(* CoDeSys 2.3.9.55 project: Test_testLib.pro *)
(* Author: Philip Henriksen *)
(* Libraries: TestLib.lib 13.6.19 08:25:14, Standard.lib 20.5.14 08:13:26, Iecsfc.lib 30.1.13 13:05:12 *)

(* PLC configuration (modules and I/O channels)
K-Bus [K_Bus] node 0, in %IB0 out %QB0 {KbusBusMode = 1; KbusCycleTime = 10000; KbusThreadPriority = 0; KbusSetOutputsToZeroOnApplicationStop = 1}
Modbus variables [PFC200MODBUS] node 1, in %IB0 out %QB0 {PlcStopBehaviour = 1; FiledbusErrorBehaviour = 1; TcpOperation = 1; TcpPort = 502; TcpTimeout = 600; UdpOperation = 1; UdpPort = 502; RtuOperation = 0; NodeId = 1; ResponseTimeout = 100; Interface = 0; Baud = 115200; StopBits = 1; Parity = 1; FlowCtrl = 0; PhysInterface = 0}
Modbus-Master [MB_MASTER] node 2, in %IB0 out %QB0
*)

(* Global variable list: Var_Constant *)
VAR_GLOBAL CONSTANT
	BTFDevice:		STRING[15] := 'Device 4194302';
END_VAR

(* Data type *)
TYPE typ_ReadProperty :
STRUCT
END_STRUCT
END_TYPE

(* POU PLC_PRG, CFC *)
PROGRAM PLC_PRG
VAR
	Test:			Fb_TestFunctionBlock;
	BoolVar:		BOOL;
	RealVar:		REAL;

	BoolOut:		BOOL;
END_VAR
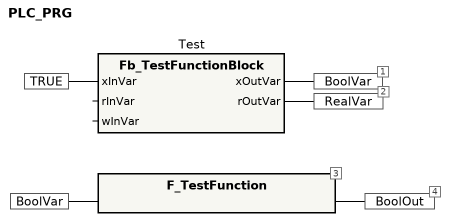
_CFC_ (* Continuous Function Chart, elements in execution order *)
#0 Test:Fb_TestFunctionBlock(xInVar: TRUE, rInVar: -, wInVar: -)
#1 BoolVar <= #0.xOutVar
#2 RealVar <= #0.rOutVar
#3 F_TestFunction(BoolVar)
#4 BoolOut <= #3
_END_CFC_
(* the same logic as Structured Text *)
Test(xInVar := TRUE);
BoolVar := Test.xOutVar;
RealVar := Test.rOutVar;
BoolOut := F_TestFunction(BoolVar);
END_PROGRAM
